RoboDK station: kr30 cnc 040219 1.rdk

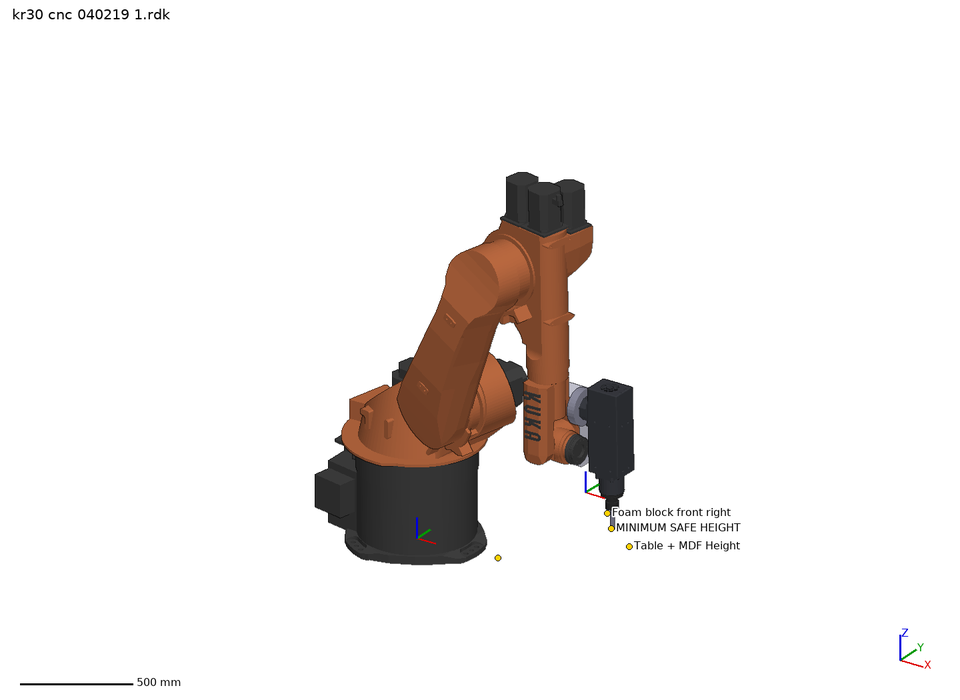
[picture v0: the station drawn from its stored meshes, robots at their saved joint values, targets as dots, program paths as lines]
Station kr30 cnc 040219 1. Poses are relative to the parent item; angles as X-Y-Z fixed-axis rotations.
  - frame KUKA KR 30 HA Base at (0, 0, 0) mm
    - robot KUKA KR 30 HA: 6 axes, payload 30 kg, reach 2033 mm, repeatability 0.05 mm, weight 665 kg
        modified DH rows (alpha deg, a mm, theta deg, d mm): 0, 0, 0, 815; -90, 350, 0, 0; 0, 850, -90, 0; -90, 145, 0, 820; 90, 0, 0, 0; -90, 0, 180, 170
        joint limits [-185, -135, -120, -350, -119, -350] to [185, 35, 158, 350, 119, 350]; home [0, -90, 90, 0, 0, 0]; saved at [11.991, -66.475, 154.983, 11.569, -89.66, -0.427]
      - tool 1/2" End Mill TCP, TCP at (337.71, -2.2, 160.57) mm, size 692.9 x 170 x 256 mm
    - target Table + MDF Height (Cartesian target) at (1304.45, -228.98, 414.16) mm, rotated rx 74.5 ry 89.96 rz -13.2 deg; joints [-4.487, -50.987, 121.357, -92.054, -90.744, 19.577] of KUKA KR 30 HA
  - frame Milling Reference at (859.69, 72.68, 436.02) mm
    - object TABLE HEIGHT NOT YET SET at (0, -1000, 0) mm, size 1193.8 x 965.2 x 609.6 mm, geometry from welding_table.sld
    - object RhinoPart at (0, 0, 0) mm
    - target Foam block back left top (Cartesian target) at (160.86, -905.12, 83.2) mm, rotated rx 6.64 ry 88.87 rz 6.23 deg; joints [50.484, -66.053, 139.001, 51.077, -80.246, -13.321] of KUKA KR 30 HA
    - target Foam block front right top (Cartesian target) at (295.04, -254.34, 79.72) mm, rotated rx 6.53 ry 88.87 rz 6.11 deg; joints [12.265, -74.97, 156.347, 11.941, -82.683, -1.906] of KUKA KR 30 HA
    - target MINIMUM SAFE HEIGHT (Cartesian target) at (314.31, -254.34, 11.19) mm, rotated rx 6.53 ry 88.87 rz 6.11 deg; joints [11.991, -66.475, 154.983, 11.569, -89.66, -0.427] of KUKA KR 30 HA
  - machining project Machining Settings: rotZ(0) | rotX(0)*rotY(0) | rotZ(0) | onStart | onPathStart | onApproach | onPoint | onRetract | onFinish | Extruder(%1) | default | default | OutOnMov(%1) | OutOffMov(%1) | onPathFinish | M_RunCode(%1)
  - machining project RhinoPart Settings: rotZ(0) | rotX(0)*rotY(0) | roty(180) | onStart | onPathStart | onApproach | onPoint | onRetract | onFinish | SetRPM(%1) | SetTool(%1) | Extruder(%1) | default | default | OutOnMov(%1) | OutOffMov(%1) | onPathFinish | M_RunCode(%1)
  - object box at (500, 500, 500) mm, size 250 x 250 x 250 mm, geometry from box.sld
